TYPE ComRob :
STRUCT
	//~
	in		: ComRobIn;
	out		: ComRobOut;
	//~
END_STRUCT
END_TYPE

(* stored: Version 1.1.0.1, ProductVersion 3.1.4024.12
   DUT ComRob: Id {b418db13-0369-097f-0768-871f402724e3} *)
